FUNCTION_BLOCK IO_AO (* Analog output (raw = Bias + OUT * Gain, 0..65535; EN = FALSE writes 0); Backend 0 simulated, 1 local IO handle (QW, e.g. GPIOChip or PWM channel), 2 Modbus CLIENT *)
  (* Standard: 61499-2 *)
  (* Version 0.1, 2026-09-28, Project contributors, AAU Smart Production Lab *)
  PACKAGE modlib;
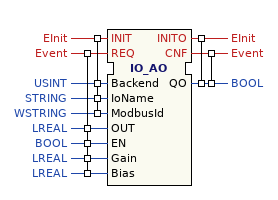
  EVENT_INPUT
    INIT : EInit WITH Backend, IoName, ModbusId;
    REQ WITH OUT, EN, Gain, Bias;
  END_EVENT
  EVENT_OUTPUT
    INITO : EInit WITH QO;
    CNF WITH QO;
  END_EVENT
  VAR_INPUT
    Backend : USINT;
    IoName : STRING;
    ModbusId : WSTRING;
    OUT : LREAL;
    EN : BOOL;
    Gain : LREAL := 1.0;
    Bias : LREAL;
  END_VAR
  VAR_OUTPUT
    QO : BOOL;
  END_VAR
  FBS
    Route : modlib::IO_RouteAO;
    Local : eclipse4diac::io::QW;
    Bus : iec61499::net::CLIENT_1_0;
  END_FBS
  EVENT_CONNECTIONS
    INIT TO Route.INIT;
    Route.INIT_IO TO Local.INIT;
    Local.INITO TO Bus.INIT;
    Bus.INITO TO Route.IO_READY;
    Route.INITO TO INITO;
    REQ TO Route.REQ;
    Route.REQ_G TO Local.REQ;
    Route.REQ_M TO Bus.REQ;
    Local.CNF TO Route.CNF_G;
    Bus.CNF TO Route.CNF_M;
    Route.CNF TO CNF;
  END_CONNECTIONS
  DATA_CONNECTIONS
    Backend TO Route.Backend;
    IoName TO Local.PARAMS;
    ModbusId TO Bus.ID;
    Route.GQI TO Local.QI;
    Route.MQI TO Bus.QI;
    Local.QO TO Route.QO_G;
    Bus.QO TO Route.QO_M;
    Route.QO TO QO;
    OUT TO Route.OUT;
    EN TO Route.EN;
    Gain TO Route.Gain;
    Bias TO Route.Bias;
    Route.Value TO Local.OUT;
    Route.Value TO Bus.SD_1;
  END_CONNECTIONS
END_FUNCTION_BLOCK
